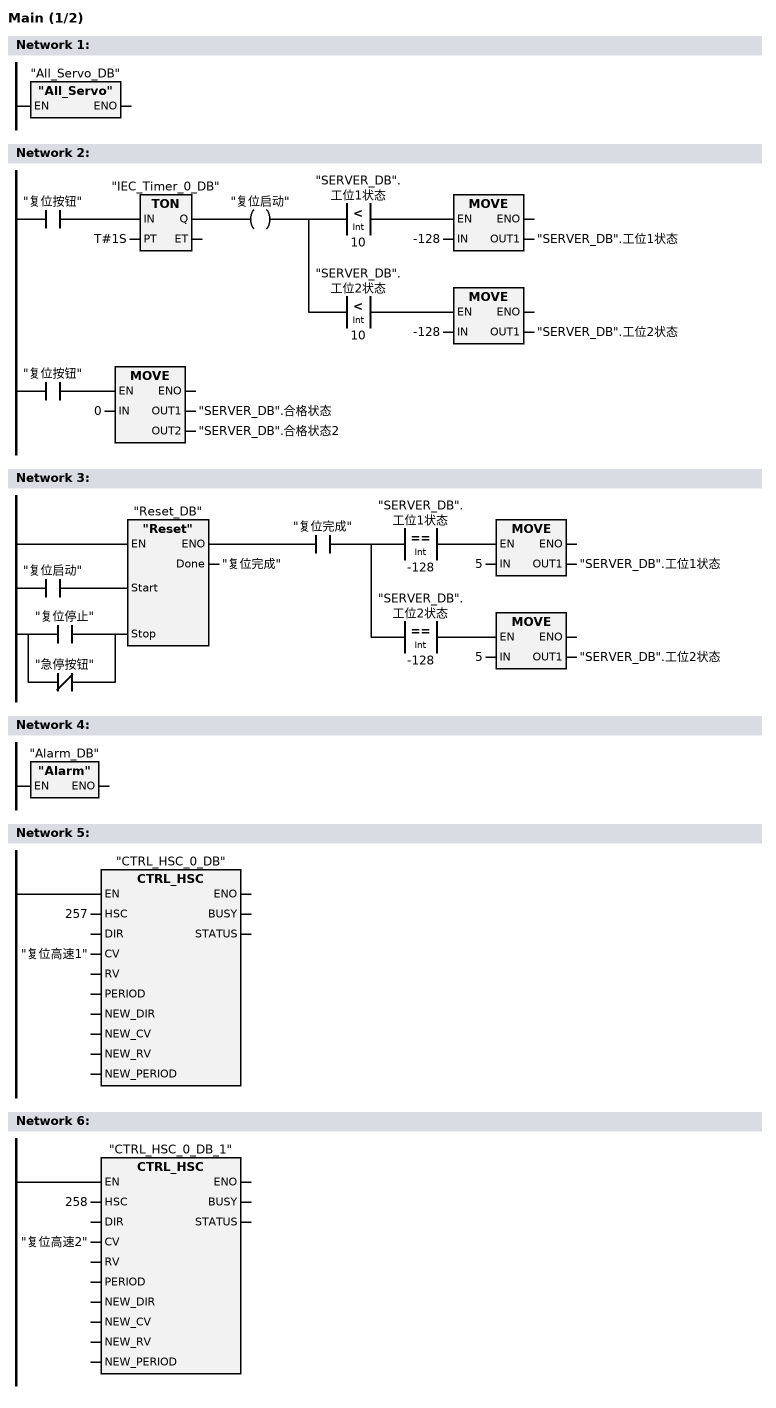
   RUNG wire#powerrail
      "All_Servo_DB"()
   END_RUNG
   // the same network as SCL:
   "All_Servo_DB"();   // "All_Servo"
END_REGION

REGION Network 2
   "IEC_Timer_0_DB".TON(IN := "复位按钮", PT := T#1S);
   "复位启动" := "IEC_Timer_0_DB".Q;
   IF "IEC_Timer_0_DB".Q AND ("SERVER_DB".工位1状态 < 10) THEN "SERVER_DB".工位1状态 := -128; END_IF;
   IF "IEC_Timer_0_DB".Q AND ("SERVER_DB".工位2状态 < 10) THEN "SERVER_DB".工位2状态 := -128; END_IF;
   IF "复位按钮" THEN
       "SERVER_DB".合格状态 := 0;
       "SERVER_DB".合格状态2 := 0;
   END_IF;
END_REGION

REGION Network 3
   RUNG wire#powerrail
      "Reset_DB"(Start := wire#w1, Stop := wire#w2, Done => "复位完成")
      Contact( "复位完成" )
      wire#w3
      { S7_Templates := "SrcType := Int" } EQ_Contact(in1 := "SERVER_DB".工位1状态, in2 := -128)
      Move(in := 5, out1 => "SERVER_DB".工位1状态)
   END_RUNG
   RUNG wire#powerrail
      Contact( "复位启动" )
   END_RUNG wire#w1
   RUNG wire#powerrail
      Contact( "复位停止" )
   END_RUNG wire#w2
   RUNG wire#powerrail
      I_Contact( "急停按钮" )
   END_RUNG wire#w2
   RUNG wire#w3
      { S7_Templates := "SrcType := Int" } EQ_Contact(in1 := "SERVER_DB".工位2状态, in2 := -128)
      Move(in := 5, out1 => "SERVER_DB".工位2状态)
   END_RUNG
   // the same network as SCL:
   "Reset_DB"(Start := "复位启动", Stop := "复位停止" OR NOT "急停按钮", Done => "复位完成", ENO => #_w1);   // "Reset"
   #_w2 := #_w1 AND "复位完成";
   IF #_w2 AND ("SERVER_DB".工位1状态 = (-128)) THEN "SERVER_DB".工位1状态 := 5; END_IF;
   IF #_w2 AND ("SERVER_DB".工位2状态 = (-128)) THEN "SERVER_DB".工位2状态 := 5; END_IF;
END_REGION

REGION Network 4
   RUNG wire#powerrail
      "Alarm_DB"()
   END_RUNG
   // the same network as SCL:
   "Alarm_DB"();   // "Alarm"
END_REGION

REGION Network 5
   "CTRL_HSC_0_DB"(HSC := 257, CV := "复位高速1");   // CTRL_HSC
END_REGION

REGION Network 6
   "CTRL_HSC_0_DB_1"(HSC := 258, CV := "复位高速2");   // CTRL_HSC
END_REGION

REGION Network 7
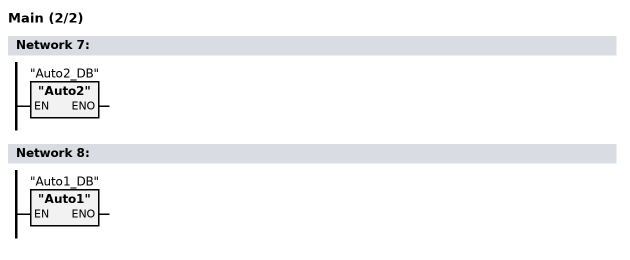
   RUNG wire#powerrail
      "Auto2_DB"()
   END_RUNG
   // the same network as SCL:
   "Auto2_DB"();   // "Auto2"
END_REGION

REGION Network 8
   RUNG wire#powerrail
      "Auto1_DB"()
   END_RUNG
   // the same network as SCL:
   "Auto1_DB"();   // "Auto1"
END_REGION
END_ORGANIZATION_BLOCK

ORGANIZATION_BLOCK "Cyclic interrupt"   // OB30, LAD, CyclicInterrupt
{ S7_Optimized_Access := 'TRUE' }
VERSION : 0.1
   VAR_INPUT
      Initial_Call : Bool;   // Initial call of this OB
      Event_Count : Int;   // Events discarded
   END_VAR
   VAR_TEMP   // added for the SCL form of the ladder/FBD networks
      _w1 : Bool;
   END_VAR
BEGIN

REGION Network 1
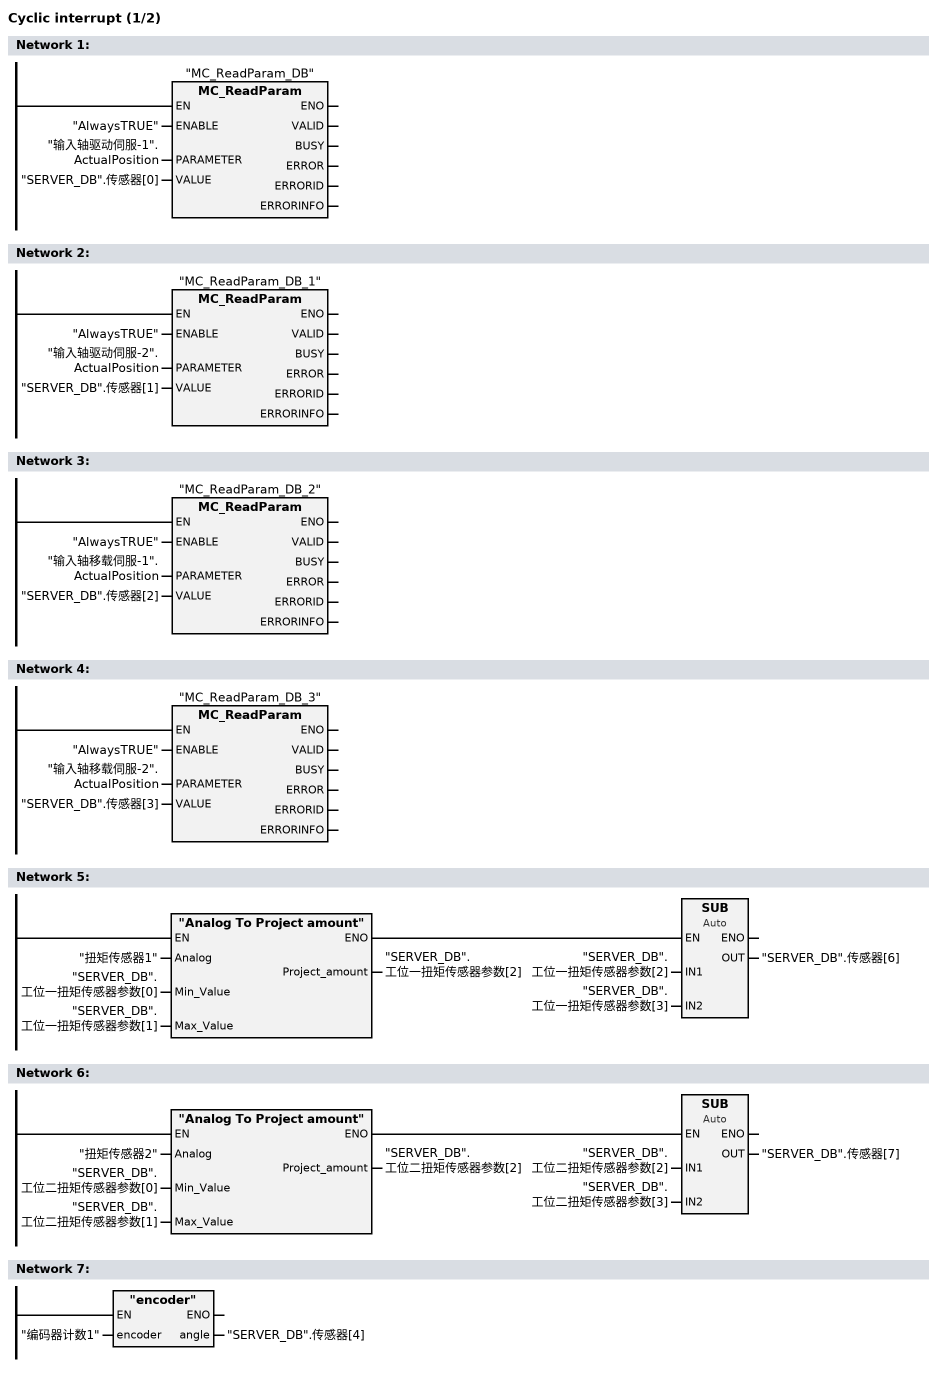
   "MC_ReadParam_DB"(Enable := "AlwaysTRUE",   // MC_ReadParam
                     Parameter := "输入轴驱动伺服-1".ActualPosition,
                     Value := "SERVER_DB".传感器[0]);
END_REGION

REGION Network 2
   "MC_ReadParam_DB_1"(Enable := "AlwaysTRUE",   // MC_ReadParam
                       Parameter := "输入轴驱动伺服-2".ActualPosition,
                       Value := "SERVER_DB".传感器[1]);
END_REGION

REGION Network 3
   "MC_ReadParam_DB_2"(Enable := "AlwaysTRUE",   // MC_ReadParam
                       Parameter := "输入轴移载伺服-1".ActualPosition,
                       Value := "SERVER_DB".传感器[2]);
END_REGION

REGION Network 4
   "MC_ReadParam_DB_3"(Enable := "AlwaysTRUE",   // MC_ReadParam
                       Parameter := "输入轴移载伺服-2".ActualPosition,
                       Value := "SERVER_DB".传感器[3]);
END_REGION

REGION Network 5
   RUNG wire#powerrail
      "Analog To Project amount"(Analog := "扭矩传感器1", Min_Value := "SERVER_DB".工位一扭矩传感器参数[0], Max_Value := "SERVER_DB".工位一扭矩传感器参数[1], Project_amount => "SERVER_DB".工位一扭矩传感器参数[2])
      Sub(in1 := "SERVER_DB".工位一扭矩传感器参数[2], in2 := "SERVER_DB".工位一扭矩传感器参数[3], out => "SERVER_DB".传感器[6])
   END_RUNG
   // the same network as SCL:
   "Analog To Project amount"(Analog := "扭矩传感器1",
                           Min_Value := "SERVER_DB".工位一扭矩传感器参数[0],
                           Max_Value := "SERVER_DB".工位一扭矩传感器参数[1],
                           Project_amount => "SERVER_DB".工位一扭矩传感器参数[2],
                           ENO => #_w1);
   IF #_w1 THEN "SERVER_DB".传感器[6] := "SERVER_DB".工位一扭矩传感器参数[2] - "SERVER_DB".工位一扭矩传感器参数[3]; END_IF;
END_REGION

REGION Network 6
   RUNG wire#powerrail
      "Analog To Project amount"(Analog := "扭矩传感器2", Min_Value := "SERVER_DB".工位二扭矩传感器参数[0], Max_Value := "SERVER_DB".工位二扭矩传感器参数[1], Project_amount => "SERVER_DB".工位二扭矩传感器参数[2])
      Sub(in1 := "SERVER_DB".工位二扭矩传感器参数[2], in2 := "SERVER_DB".工位二扭矩传感器参数[3], out => "SERVER_DB".传感器[7])
   END_RUNG
   // the same network as SCL:
   "Analog To Project amount"(Analog := "扭矩传感器2",
                           Min_Value := "SERVER_DB".工位二扭矩传感器参数[0],
                           Max_Value := "SERVER_DB".工位二扭矩传感器参数[1],
                           Project_amount => "SERVER_DB".工位二扭矩传感器参数[2],
                           ENO => #_w1);
   IF #_w1 THEN "SERVER_DB".传感器[7] := "SERVER_DB".工位二扭矩传感器参数[2] - "SERVER_DB".工位二扭矩传感器参数[3]; END_IF;
END_REGION

REGION Network 7
   RUNG wire#powerrail
      "encoder"(encoder := "编码器计数1", angle => "SERVER_DB".传感器[4])
   END_RUNG
   // the same network as SCL:
   "encoder"(encoder := "编码器计数1", angle => "SERVER_DB".传感器[4]);
END_REGION

REGION Network 8
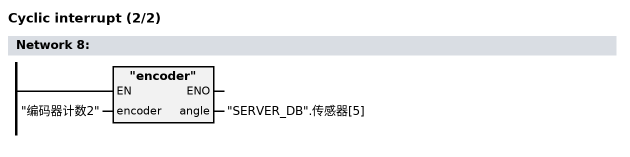
   RUNG wire#powerrail
      "encoder"(encoder := "编码器计数2", angle => "SERVER_DB".传感器[5])
   END_RUNG
   // the same network as SCL:
   "encoder"(encoder := "编码器计数2", angle => "SERVER_DB".传感器[5]);
END_REGION
END_ORGANIZATION_BLOCK